{attribute 'GeneratedUsingTerminal: EL5102-0000-0016'}
{attribute addProperty BoxType "EL5102-0000-0016"}
{attribute addProperty Id "ControlAT %Q*Control_D4F3D88010Set_counter_valueAT %Q*UDINT4"}
{attribute addProperty CRC "1284141973"}
{attribute addProperty Size "14"}
TYPE ENC_Control_Channel_4C8A7395 :
STRUCT
	{attribute addProperty Name "Control"}
	Control AT %Q* : Control_D4F3D880;
	{attribute addProperty Name "Set_counter_value"}
	Set_counter_value AT %Q* : UDINT;
END_STRUCT
END_TYPE

(* stored: Version 1.2.0.0, ProductVersion 3.1.4024.9
   DUT ENC_Control_Channel_4C8A7395: Id {961f3891-e8f2-46e2-a196-5ae222670308} *)
